{attribute 'qualified_only'}
{attribute 'strict'}
TYPE E_Status :
(
	NotReady,
	Ready,
	Starting,
	Running,
	Stopping,
	Fault,
	Joystick
);
END_TYPE

(* stored: Version 1.1.0.1, ProductVersion 3.1.4024.12
   DUT E_Status: Id {28274fdb-23c6-4366-8cdc-47c2e283b658} *)
